Staubli VAL3: blow.pgx

program blow()
begin
  // This program set the Blow of the tool for _nBlowDelay seconds.
  //
  // Input parameters
  //  None            :
  //
  // Output parameters
  //  None            :
  //
  //----------------------------------------------------------------
  //
  do
    wait(_nBlowDelay>0)
    dVacuum=false
    dBlow=true
    delay(_nBlowDelay)
    dBlow=false
    _nBlowDelay=0
    delay(0)
  until false
end
